{attribute 'linkalways'} 
{attribute 'no_explicit_call' := 'This FB is a CLASS and must be accessed using methods or properties'}
{attribute 'enable_dynamic_creation'}
FUNCTION_BLOCK FINAL GT_LWORD EXTENDS Node
VAR
	in1 : _LWORD(0);
	in2 : _LWORD(0);
	out : _BOOL(FALSE);
END_VAR

METHOD PUBLIC Clone : I_Node
VAR
	pNode : POINTER TO GT_LWORD;
END_VAR
pNode := __NEW(GT_LWORD);
Clone := pNode^;
END_METHOD

METHOD FB_init : BOOL
VAR_INPUT
	bInitRetains : BOOL; // if TRUE, the retain variables are initialized (warm start / cold start)
	bInCopyCode : BOOL;  // if TRUE, the instance afterwards gets moved into the copy code (online change)
END_VAR
AddInput('in1',THIS^.in1);
AddInput('in2',THIS^.in2);
AddOutput('out', THIS^.out);
END_METHOD

METHOD PROTECTED OnExecute
VAR
END_VAR
out.Value := in1.Value > in2.Value;
END_METHOD

END_FUNCTION_BLOCK

(* stored: Version 1.1.0.1, ProductVersion 3.1.4024.15
   POU GT_LWORD: Id {b975d2b6-9835-445e-927b-0a00e4a3db05}, SpecialFunc None
   Folder Constructor: Id {af813005-135a-4e68-adbb-ee046cdd6799}
   Method Clone: Id {f4fb1008-7a6b-47d8-a88d-46014ea61357}
   Method FB_init: Id {c2ac0c68-ef36-4e2f-b156-d2eb47e93d31}
   Method OnExecute: Id {8872bbc4-af90-490d-825f-f9cb5166b8b3} *)
